FUNCTION_BLOCK AutoSamplar (* Composite Function Block Type *)
  (* Standard: 61499-2 *)
  (* Version 0.0, 9/26/2024, SESA713705, Schneider Electric, template *)
  PACKAGE SE.Nereda;
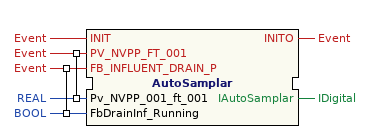
  EVENT_INPUT
    INIT;
    PV_NVPP_FT_001 WITH Pv_NVPP_001_ft_001;
    FB_INFLUENT_DRAIN_P WITH FbDrainInf_Running;
  END_EVENT
  EVENT_OUTPUT
    INITO;
  END_EVENT
  VAR_INPUT
    Pv_NVPP_001_ft_001 : REAL;
    FbDrainInf_Running : BOOL;
  END_VAR
  PLUGS
    IAutoSamplar : IDigital;
  END_PLUGS
  (* 01 - FUNCTIONAL INPUT INTERFACE *)
  (* 00 - INITIALIZATION *)
  (* 02 - FUNCTIONNAL OUTPUT INTERFACE *)
  (* 05 - LOGIC *)
  (* HMI *)
  (* Auto Samplar Logic *)
  (* Delay *)
  (* Check if Flow >= Flow Sp (HMI) *)
  (* Calculate the 1 metre cube from the Flow *)
  FBS
    IThis : AutoSamplar_HMI(QI := TRUE);
    AutoSamplar_Logic : AutoSamplar_Manager;
    Pulse : E_DELAY(DT := T#500ms);
    FlowCompare : COMPARE_1329C2AB45109BAAB; {SET_ATTRIBUTE(Configuration.GenericFBType.InterfaceParams, Runtime.Standard#CNT:=2;IN${CNT$}:REAL)}
    MetreCubeTime_Calculator : MetreCubeTime_Calculator;
    DelayTime : E_DELAY_V_D;
    Counte_1m_Cube : E_DELAY_V_D;
    FlowIsOK : boolValueChanged;
    REAL2TIME : REAL2TIME;
    PulseCmd : boolValueChanged;
    CmdPulse : BOOL2INT;
    FlowSmooth : RealValueChanged;
    Counte1mCube : E_DELAY_V;
    PulseCounter : CountPulse;
  END_FBS
  EVENT_CONNECTIONS
    PV_NVPP_FT_001 TO FlowCompare.REQ;
    DelayTime.INITO TO Counte_1m_Cube.INIT;
    Counte_1m_Cube.INITO TO INITO;
    Counte_1m_Cube.INITO TO AutoSamplar_Logic.INIT;
    Counte1mCube.49657F677FC47D45 TO AutoSamplar_Logic.REQ_1M_CUBE_DONE;
    DelayTime.1457E63E0C241C83 TO AutoSamplar_Logic.REQ_DELAY_TIME_DONE;
    Pulse.EO TO AutoSamplar_Logic.REQ_PULSE_DELAY;
    FB_INFLUENT_DRAIN_P TO AutoSamplar_Logic.REQ_INF_PUMP_ON;
    FlowCompare.CNF TO FlowIsOK.REQ;
    FlowIsOK.CHD TO AutoSamplar_Logic.REQ_FLOW_SP_IS_OK;
    PV_NVPP_FT_001 TO FlowSmooth.77F8F9CFF707DAFF;
    MetreCubeTime_Calculator.CNF_TIME TO REAL2TIME.9954577AA24F9DD6;
    AutoSamplar_Logic.CNF_CYCLE TO Counte1mCube.73DC624F4AA9B9EF;
    AutoSamplar_Logic.CNF_DELAY_TIME TO DelayTime.START;
    AutoSamplar_Logic.CNF_DELAY_PULSE TO Pulse.START;
    AutoSamplar_Logic.CNF_PULSE TO PulseCmd.REQ;
    PulseCmd.CHD TO CmdPulse.DD5870AA881150BB;
    CmdPulse.6FC99A5BD1C38561 TO IAutoSamplar.REQ;
    FlowSmooth.93AE3729A9342678 TO MetreCubeTime_Calculator.REQ_FLOW;
    AutoSamplar_Logic.CNF_CYCLE TO Counte_1m_Cube.START;
    PulseCmd.CHD TO PulseCounter.37F2B181FA61BC7D;
    INIT TO IThis.9E2D5FD52A41FA97;
    PulseCmd.CHD TO IThis.E9347DD12F47CD58;
    PulseCounter.EEBF1C26172F0C71 TO IThis.E9347DD12F47CD58;
    AutoSamplar_Logic.CNF_STATE TO IThis.B538FB3EA4FE2B16;
    Counte_1m_Cube.INITO TO IThis.4ECDB5B072C1C4D7;
    REAL2TIME.79B40746AB555956 TO IThis.600FCA08E43F4544;
    IThis.15445CD6D7538879 TO DelayTime.INIT;
    IThis.113EB47D18B327BE TO DelayTime.START;
    IThis.334B88A0D5C84CD1 TO FlowCompare.REQ;
  END_CONNECTIONS
  DATA_CONNECTIONS
    Pv_NVPP_001_ft_001 TO FlowCompare.IN1;
    FlowCompare.GE TO FlowIsOK.Input;
    FlowIsOK.Output TO AutoSamplar_Logic.FlowSp_IsOK;
    FbDrainInf_Running TO AutoSamplar_Logic.InfluentDrainPumpON;
    Pv_NVPP_001_ft_001 TO FlowSmooth.25B5287A5784F3EC;
    REAL2TIME.8AC404843F53B283 TO Counte1mCube.EA75F27E53BC78A7;
    MetreCubeTime_Calculator.MetreCube_Time TO REAL2TIME.158B8AA7B31D2617;
    AutoSamplar_Logic.Pulse TO PulseCmd.Input;
    PulseCmd.Output TO CmdPulse.4573FC8F228EB71D;
    CmdPulse.A6DEF5F9C27C1848 TO IAutoSamplar.Value;
    Counte1mCube.A0AC39E38E6A8452 TO AutoSamplar_Logic.32D95873A2868127;
    FlowSmooth.AA81B8787A42C5C8 TO MetreCubeTime_Calculator.FlowPv;
    REAL2TIME.8AC404843F53B283 TO Counte_1m_Cube.DT1;
    PulseCmd.Output TO PulseCounter.3EFE041B4A3DB1DD;
    PulseCmd.Output TO IThis.75FBC455C9E40C8C;
    AutoSamplar_Logic.State TO IThis.3CCCBB1B7B75B659;
    REAL2TIME.8AC404843F53B283 TO IThis.C0897FF52680C92B;
    Pv_NVPP_001_ft_001 TO IThis.2DA02A18EF91EF18;
    IThis.2202B95F15A70903 TO DelayTime.DT1;
    IThis.E66076390A5B5835 TO FlowCompare.IN2;
    PulseCounter.5B7001294FCB7A80 TO IThis.9301876BE9349110;
  END_CONNECTIONS
END_FUNCTION_BLOCK
